TYPE Type_ModuleCommIn_Drilling :
STRUCT
	m_Work					:BOOL;
	m_OutOfArea				:BOOL;
	m_PartDropped			:BOOL;
END_STRUCT
END_TYPE

(* stored: Version 1.1.0.1, ProductVersion 3.1.4024.3
   DUT Type_ModuleCommIn_Drilling: Id {e1d1db2b-8323-43f4-a06c-06f8a1e1cad0} *)
